ABB RobotStudio station: FigurDrawV7.5CodeDone.rspag

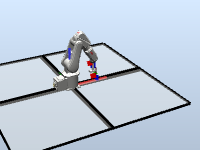
--- station ---
Station Ny63 (saved by RobotStudio 6.8.8307.1040)
Controller 120-100761
  mechanical unit ROB_1: IRB120_3_58__01, 6 joints, base frame (0, 0, 0) mm
Layout (positions relative to the parent item):
  - IRB120_3_58__01 [mechanism, from Robots\IRB120_3_58_G_01.rslib] at (0, 0, 0) mm; joint values [0, 0.3343, 0.705, 0, 0.5315, 0] (rad or m)
  - Tusch3 [mechanism, from Libraries\Tusch3.rslib] at (302, 0, 248.2) mm, rotated rx 180 ry 0 rz 180 deg
Attachment: Tusch3 is attached to IRB120_3_58__01 / Link6

--- Backups/120-100761/RAPID/TASK1/PROGMOD/CalibData.mod ---
MODULE CalibData
	PERS tooldata Tusch3:=[TRUE,[[-40.7,0,181.64],[1,0,0,0]],[0.6,[14,0,78.3],[1,0,0,0],0.007,0.01,0.01]];
ENDMODULE

--- Backups/120-100761/RAPID/TASK1/PROGMOD/MainModule.mod ---
MODULE MainModule
    PERS num nAntal:=0;
    PERS num nType:=0;
    PERS num varZ:=0;
    PERS num varZCounter:=0;
    PERS num varX:=0;
    PERS num varY:=0;
    !CONST robtarget UdgangPos:=[[342.70,0.00,376.36],[5.8086E-8,0,-1,0],[0,0,0,0],[9E+9,9E+9,9E+9,9E+9,9E+9,9E+9]];
	PERS robtarget p20:=[[342.70,0.00,0.56],[5.94159E-8,2.65924E-30,1,2.10468E-31],[0,0,0,0],[9E+9,9E+9,9E+9,9E+9,9E+9,9E+9]];
	!PERS robtarget p30:=[[342.70,200.28,0.56],[1.19502E-7,6.67535E-8,1,2.45704E-8],[0,-1,0,0],[9E+9,9E+9,9E+9,9E+9,9E+9,9E+9]];
	!PERS robtarget p40:=[[550.25,200.28,0.56],[6.16107E-8,-1.77398E-8,1,-1.12879E-8],[0,-1,0,0],[9E+9,9E+9,9E+9,9E+9,9E+9,9E+9]];
	!PERS robtarget p50:=[[550.25,-274.17,0.56],[1.20042E-7,6.79573E-9,1,-3.03003E-8],[-1,0,-1,0],[9E+9,9E+9,9E+9,9E+9,9E+9,9E+9]];
	!PERS robtarget p60:=[[345.29,-274.17,0.56],[1.63644E-8,3.67595E-8,1,3.67745E-8],[-1,0,-1,0],[9E+9,9E+9,9E+9,9E+9,9E+9,9E+9]];
    !PERS robtarget p70:=[[342.70,-0.00,0.56],[5.94159E-8,2.65924E-30,1,2.10468E-31],[0,0,0,0],[9E+9,9E+9,9E+9,9E+9,9E+9,9E+9]];
    PERS robtarget p80:=[[342.70,-0.00,0.56],[5.94159E-8,2.65924E-30,1,2.10468E-31],[0,0,0,0],[9E+9,9E+9,9E+9,9E+9,9E+9,9E+9]];


    PROC main()
        IF nType = 1 THEN
            cirkel;
        ELSEIF nType = 2 THEN
            firekant;
        ELSEIF nType = 3 THEN
            trekant;
        ENDIF
	ENDPROC

    PROC cirkel() !Kode for Cirkel, og de antal den skal køre.
        nType:=0; !nulstillet Type Tallet.
        varZCounter:= varZ; !Sætter ny højde den skal starte på.
        MoveL  Offs(p20,0,0,varZcounter), v1000, fine, Tusch3; !udgangspunkt før den laver Cirkel.
        FOR i FROM 0 TO nAntal DO !For Loop, fra en til "nAntal" DO
            TPErase; !Sletter TPErease for at kunne skrive igen.
            !TPWrite "Laver Cirkel"; !Skriver "Laver Cirkkel".
            MoveC Offs(p20,100,100,varZCounter), Offs(p80,200,0,varZCounter), v1000, fine, Tusch3; !Første halvdel af Cirklen.
            MoveC Offs(p20,100,-100,varZCounter), Offs(p80,0,0,varZCounter), v1000, fine, Tusch3; !Anden halvdel af Cirklen.
            varZCounter:= varZCounter+varZ;
            MoveL  Offs(p20,0,0,varZCounter), v1000, fine, Tusch3; !udgangspunkt før den laver Cirkel.
        ENDFOR!Kodeslut For Loop.
        varZCounter:=0;!varZCounter af routine Value bliver nulstillet med tallet 0.
        varZ:=0; !varZ af routine Value bliver nulstillet med tallet 0.
        nAntal:=0; !Antal af routine Value bliver nulstillet med tallet 0.
        !MoveL UdgangPos, v1000, z50, Tusch3; !Udgangspunkt
	ENDPROC!Kodeslut Cirkel.

    PROC firekant() !Kode for Firekant, og de antal den skal køre. Samme kommentar ovenover.
        nType:=0; !nulstillet Type Tallet.
        varZCounter:= varZ; !Sætter ny højde den skal starte på.
        MoveL  Offs(p20,0,0,varZCounter), v1000, fine, Tusch3; !udgangspunkt før den laver firekant.
        FOR i FROM 0 TO nAntal DO
            TPErase;
            !TPWrite "Laver Firekant";
            MoveL Offs(p20,varY,0,varZCounter), v1000, fine, Tusch3;
            MoveL Offs(p20,varY,varX,varZCounter), v1000, fine, Tusch3;
            MoveL Offs(p20,varY,varX,varZCounter), v1000, fine, Tusch3;
            MoveL Offs(p20,0,varX,varZCounter), v1000, fine, Tusch3;
            MoveL Offs(p20,0,0,varZCounter), v1000, fine, Tusch3;
            varZCounter:= varZCounter+varZ;
            !En ANDEN MÅDE AT LAVE FIREKANT PÅ.
            !MoveL p30, v1000, fine, Tusch3;
            !MoveL p40, v1000, fine, Tusch3;
            !MoveL p50, v1000, fine, Tusch3;
            !MoveL p60, v1000, fine, Tusch3;
            !MoveL p70, v1000, fine, Tusch3;
            MoveL  Offs(p20,0,0,varZCounter), v1000, fine, Tusch3; !udgangspunkt før den laver firekant.
        ENDFOR
        varZCounter:=0;!varZCounter af routine Value bliver nulstillet med tallet 0.
        varX:=0;
        varY:=0;
        varZ:=0; !varZ af routine Value bliver nulstillet med tallet 0.
        nAntal:=0; !Antal af routine Value bliver nulstillet med tallet 0.
        !MoveL UdgangPos, v1000, z50, Tusch3; !Udgangspunkt
	ENDPROC

    !PROC Rektangel() !Kode for Rektangel, og de antal den skal køre. Samme kommentar ovenover.
       !nType:=0; !nulstillet Type Tallet.
        !varZCounter:= varZ; !Sætter ny højde den skal starte på.
        !MoveL  Offs(p20,0,0,varZCounter), v1000, fine, Tusch3; !udgangspunkt før den laver rektangel.
        !FOR i FROM 0 TO nAntal DO
            !TPErase;
            !TPWrite "Laver Rektangel";
            !MoveL Offs(p30,0,0,varZCounter), v1000, fine, Tusch3;
            !MoveL Offs(p40,0,0,varZCounter), v1000, fine, Tusch3;
            !MoveL Offs(p50,0,0,varZCounter), v1000, fine, Tusch3;
            !MoveL Offs(p60,0,0,varZCounter), v1000, fine, Tusch3;
            !MoveL Offs(p70,0,0,varZCounter), v1000, fine, Tusch3;
            !varZCounter:= varZCounter+varZ;
            !MoveL Offs(p20,0,0,varZCounter), v1000, fine, Tusch3; !udgangspunkt før den laver rektangel

        !ENDFOR
        !varX:=0;
        !varY:=0;
        !varZCounter:=0;!varZCounter af routine Value bliver nulstillet med tallet 0.
        !varZ:=0; !varZ af routine Value bliver nulstillet med tallet 0.
        !nAntal:=0; !Antal af routine Value bliver nulstillet med tallet 0.
        !MoveL UdgangPos, v1000, z50, Tusch3; !Udgangspunk
	!ENDPROC

    PROC trekant() !Kode for trekant, og de antal den skal køre. Samme kommentar ovenover.
        nType:=0; !nulstillet Type Tallet.
        varZCounter:= varZ; !Sætter ny højde den skal starte på.
        MoveL  Offs(p20,0,0,varZCounter), v1000, fine, Tusch3; !udgangspunkt før den laver firekant.
        FOR i FROM 0 TO nAntal DO
            TPErase;
            !TPWrite "Laver trekant";
            MoveL Offs(p20,varY,0,varZCounter), v1000, fine, Tusch3;
            MoveL Offs(p20,varY,varX,varZCounter), v1000, fine, Tusch3;
            !MoveL Offs(p20,varY,varX,varZCounter), v1000, fine, Tusch3;
            MoveL  Offs(p20,0,0,varZCounter), v1000, fine, Tusch3;
            varZCounter:= varZCounter+varZ;
            MoveL  Offs(p20,0,0,varZCounter), v1000, fine, Tusch3; !udgangspunkt før den laver trekant.
        ENDFOR
        varZCounter:=0;!varZCounter af routine Value bliver nulstillet med tallet 0.
        varX:=0;
        varY:=0;
        varZ:=0; !varZ af routine Value bliver nulstillet med tallet 0.
        nAntal:=0; !Antal af routine Value bliver nulstillet med tallet 0.
        !MoveL UdgangPos, v1000, z50, Tusch3; !Udgangspunkt
	ENDPROC

ENDMODULE

--- Backups/120-100761/RAPID/TASK1/SYSMOD/LINKEDM.sys ---
%%%
  VERSION:1
  LANGUAGE:ENGLISH
%%%

MODULE LINKEDM (SYSMODULE)

! FOLLOWER
!     Name of electronically linked follower axis used by operator at teach pendent.
      PERS string l_f_axis_name{5}       :=  ["",  "", "", "", ""];

!     Name of the mechanical unit for follower axis.
      PERS string l_f_mecunt_n{5}  :=  ["", "", "", "", ""];

!     Linked follower axis number in the mechanical unit (first axis in mech. unit is number 1).
      PERS num l_f_axis_no{5}      :=  [0,          0,   0,  0,  0];

! MASTER
!     Name of the mechanical unit for linked master axis.
      PERS string l_m_mecunt_n{5} :=  ["", "", "", "", ""];

!     Linked master axis number in the mechanical unit (first axis in mech. unit is number 1).
!     See axis number table in documentation for different master mechanical units.
      PERS num l_m_axis_no{5}     :=  [0,  0,  0,  0,  0];

! POSITION OFFSET
!     The increase of the allowed offset position between the master and follower
!     positions, used when starting AUTO mode. As soon as the offset is decreased
!     the old configurated parameter is used.
!     Example: 3 => the configurated value of allowed offset is increased 3 times.
      PERS num offset_ratio{5}       :=  [10,  10,   10,  10,  10];

! SPEED RATIO
!     Speed_ratio used in AUTO and JOG modes [ very_slow   slow    normal    fast]
!     Value 1 = max allowed manual speed.
      CONST num speed_ratio {20}      := [0.01, 0.01, 0.01, 0.01, 0.01,
                                          0.05, 0.05, 0.05, 0.05, 0.05,
                                          0.20, 0.20, 0.20, 0.20, 0.20,
                                          1.00, 1.00, 1.00, 1.00, 1.00];

! STEP SIZE
!     Displacement position used in JOG mode for each activation of positive or
!     negative movement.                  [very_short    short   normal   long]
!     Unit degees or meter.
      CONST num displacement {20}     := [0.001, 0.001, 0.001, 0.001, 0.001,
                                          0.005, 0.005, 0.005, 0.005, 0.005,
                                          0.020, 0.020, 0.020, 0.020, 0.020,
                                          0.100, 0.100, 0.100, 0.100, 0.100];


!-------------------------------------------------------------
 PROC Linked_m ()
      Linked_m_exe ;
 ENDPROC
ENDMODULE

--- Backups/120-100761/HOME/Ja1program/MainModule.mod ---
MODULE MainModule
	CONST robtarget Udgpos:=[[346.14,-2.47,470.78],[0.0835884,0.0167447,-0.995045,0.0511663],[0,-1,0,0],[9E+09,9E+09,9E+09,9E+09,9E+09,9E+09]];
	PROC main()
		MoveJ Udgpos, v1000, z50, tool0;
	ENDPROC
ENDMODULE

--- Backups/120-100761/HOME/Spids/MainModule.mod ---
MODULE MainModule
	PROC main()
        <SMT>
	ENDPROC
ENDMODULE

--- Backups/120-100761/SYSPAR/EIO.cfg ---
EIO:CFG_1.0:6:1::
#
INDUSTRIAL_NETWORK:

      -Name "DeviceNet" -Label "DeviceNet Master/Slave Network" -Address "2"
#
DEVICENET_DEVICE:

      -Name "D652_10" -VendorName "ABB Robotics" -ProductName "24 VDC Unit"\
      -Address 10 -ProductCode 26 -DeviceType 7 -ConnectionType "COS"\
      -OutputSize 2 -InputSize 2
#
DEVICENET_INTERNAL_DEVICE:

      -Name "DN_Internal_Device" -VendorName "ABB Robotics"\
      -ProductName "DeviceNet Internal Slave Device"
#
EIO_SIGNAL:

      -Name "DI10_1" -SignalType "DI" -Device "D652_10" -DeviceMap "0"\
      -Access "All"

      -Name "DI10_2" -SignalType "DI" -Device "D652_10" -DeviceMap "1"

      -Name "DI10_3" -SignalType "DI" -Device "D652_10" -DeviceMap "2"

      -Name "DI10_4" -SignalType "DI" -Device "D652_10" -DeviceMap "3"

      -Name "DI10_5" -SignalType "DI" -Device "D652_10" -DeviceMap "4"

      -Name "DI10_6" -SignalType "DI" -Device "D652_10" -DeviceMap "5"

      -Name "DI10_7" -SignalType "DI" -Device "D652_10" -DeviceMap "6"

      -Name "DI10_8" -SignalType "DI" -Device "D652_10" -DeviceMap "7"

      -Name "DI10_9" -SignalType "DI" -Device "D652_10" -DeviceMap "8"

      -Name "DI10_10" -SignalType "DI" -Device "D652_10" -DeviceMap "9"

      -Name "DI10_11" -SignalType "DI" -Device "D652_10" -DeviceMap "10"

      -Name "DI10_12" -SignalType "DI" -Device "D652_10" -DeviceMap "11"

      -Name "DI10_13" -SignalType "DI" -Device "D652_10" -DeviceMap "12"

      -Name "DI10_14" -SignalType "DI" -Device "D652_10" -DeviceMap "13"

      -Name "DI10_15" -SignalType "DI" -Device "D652_10" -DeviceMap "14"

      -Name "DI10_16" -SignalType "DI" -Device "D652_10" -DeviceMap "15"

      -Name "DO10_1" -SignalType "DO" -Device "D652_10" -DeviceMap "0"\
      -Access "All"

      -Name "DO10_2" -SignalType "DO" -Device "D652_10" -DeviceMap "1"\
      -Access "All"

      -Name "DO10_3" -SignalType "DO" -Device "D652_10" -DeviceMap "2"\
      -Access "All"

      -Name "DO10_4" -SignalType "DO" -Device "D652_10" -DeviceMap "3"\
      -Access "All"

      -Name "DO10_5" -SignalType "DO" -Device "D652_10" -DeviceMap "4"\
      -Access "All"

      -Name "DO10_6" -SignalType "DO" -Device "D652_10" -DeviceMap "5"\
      -Access "All"

      -Name "DO10_7" -SignalType "DO" -Device "D652_10" -DeviceMap "6"\
      -Access "All"

      -Name "DO10_8" -SignalType "DO" -Device "D652_10" -DeviceMap "7"\
      -Access "All"

      -Name "DO10_9" -SignalType "DO" -Device "D652_10" -DeviceMap "8"\
      -Access "All"

      -Name "DO10_10" -SignalType "DO" -Device "D652_10" -DeviceMap "9"\
      -Access "All"

      -Name "DO10_11" -SignalType "DO" -Device "D652_10" -DeviceMap "10"\
      -Access "All"

      -Name "DO10_12" -SignalType "DO" -Device "D652_10" -DeviceMap "11"\
      -Access "All"

      -Name "DO10_13" -SignalType "DO" -Device "D652_10" -DeviceMap "12"\
      -Access "All"

      -Name "DO10_14" -SignalType "DO" -Device "D652_10" -DeviceMap "13"\
      -Access "All"

      -Name "DO10_15" -SignalType "DO" -Device "D652_10" -DeviceMap "14"\
      -Access "All"

      -Name "DO10_16" -SignalType "DO" -Device "D652_10" -DeviceMap "15"\
      -Access "All"
